// TIA Portal V19 export
ORGANIZATION_BLOCK "Main"   // OB1, LAD, ProgramCycle
TITLE = "Main Program Sweep (Cycle)"
{ S7_Optimized_Access := 'TRUE' }
// stored: AutoNumber false, SetENOAutomatically false
   VAR_INPUT
      Initial_Call : Bool;   // Initial call of this OB
      Remanence : Bool;   // =True, if remanent data are available
   END_VAR
BEGIN

REGION Network 1: Map clock byte to output of dq card
   // Display "to" and "from" using move command for troubleshooting
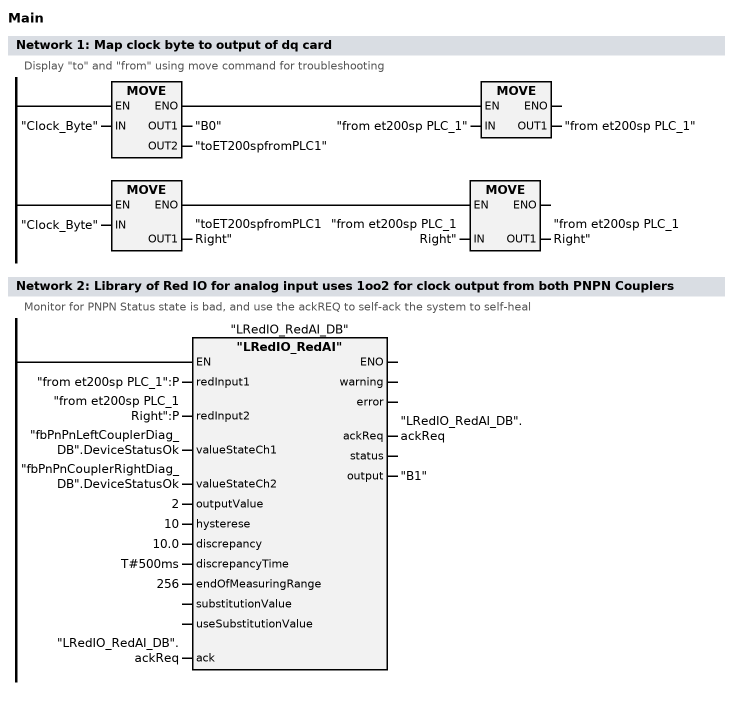
   RUNG wire#powerrail
      Move(in := "Clock_Byte", out1 => "B0", out2 => "toET200spfromPLC1")
      Move(in := "from et200sp PLC_1", out1 => "from et200sp PLC_1")
   END_RUNG
   RUNG wire#powerrail
      Move(in := "Clock_Byte", out1 => "toET200spfromPLC1 Right")
      Move(in := "from et200sp PLC_1 Right", out1 => "from et200sp PLC_1 Right")
   END_RUNG
   // the same network as SCL:
   "B0" := "Clock_Byte";
   "toET200spfromPLC1" := "Clock_Byte";
   "from et200sp PLC_1" := "from et200sp PLC_1";
   "toET200spfromPLC1 Right" := "Clock_Byte";
   "from et200sp PLC_1 Right" := "from et200sp PLC_1 Right";
END_REGION

REGION Network 2: Library of Red IO for analog input uses 1oo2 for clock output from both PNPN Couplers
   // Monitor for PNPN Status state is bad, and use the ackREQ to self-ack the system to self-heal
   RUNG wire#powerrail
      "LRedIO_RedAI_DB"(redInput1 := "from et200sp PLC_1":P, redInput2 := "from et200sp PLC_1 Right":P, valueStateCh1 := "fbPnPnLeftCouplerDiag_DB".DeviceStatusOk, valueStateCh2 := "fbPnPnCouplerRightDiag_DB".DeviceStatusOk, outputValue := 2, hysterese := 10, discrepancy := 10.0, discrepancyTime := T#500ms, endOfMeasuringRange := 256, substitutionValue :=, useSubstitutionValue :=, ack := "LRedIO_RedAI_DB".ackReq, warning =>, error =>, ackReq => "LRedIO_RedAI_DB".ackReq, status =>, output => "B1")
   END_RUNG
   // the same network as SCL:
   "LRedIO_RedAI_DB"(redInput1 := "from et200sp PLC_1":P,   // "LRedIO_RedAI"
                     redInput2 := "from et200sp PLC_1 Right":P,
                     valueStateCh1 := "fbPnPnLeftCouplerDiag_DB".DeviceStatusOk,
                     valueStateCh2 := "fbPnPnCouplerRightDiag_DB".DeviceStatusOk,
                     outputValue := 2,
                     hysterese := 10,
                     discrepancy := 10.0,
                     discrepancyTime := T#500ms,
                     endOfMeasuringRange := 256,
                     ack := "LRedIO_RedAI_DB".ackReq,
                     ackReq => "LRedIO_RedAI_DB".ackReq,
                     output => "B1");
END_REGION
END_ORGANIZATION_BLOCK
